(* Logix 5000 project; controller ICA19 vendor 1 type 14 code 150 rev 37.11; software revision 37.00 *)

TASK MainTask (continuous, watchdog 500 ms) : MainProgram

MODULES
   Local : vendor 1 type 14 code 150 (Compact 0, rev 37.11)
      Discrete_IO : Embedded (Compact 1, rev 3.1, Output RPI 20 ms)
      Analog_IO : Embedded (Compact 2, rev 1.1, Output RPI 80 ms)
      Counters : Embedded (Compact 3, rev 1.1, Output RPI 20 ms)
END_MODULES

VAR_GLOBAL   (* controller tags *)
   BottomLimit : ALIAS FOR Local:1:I.Data.1;
   Control : ALIAS FOR Local:1:I.Data.12;
   Door : STRING := 'Door is:';
   DoorClosed : STRING := 'Closed';
   DoorClosing : STRING := ' closing';
   DoorOpened : STRING := ' opening';
   DoorOpening : STRING := 'Opened';
   DoorOut : STRING;
   DoorStopped : STRING := 'stopped';
   MotorDOWN : ALIAS FOR Local:1:O.Data.0;
   MotorStop : ALIAS FOR Local:1:O.Data.2;
   MotorUP : ALIAS FOR Local:1:O.Data.1;
   Safety : STRING;
   SafetyLaser : ALIAS FOR Local:1:I.Data.11;
   SEQ : DINT;
   TopBottom : ALIAS FOR Local:1:I.Data.3;
   TopLimit : ALIAS FOR Local:1:I.Data.2;
END_VAR

PROGRAM MainProgram   (* main routine MainRoutine *)

ROUTINE MainRoutine   (* ladder *)
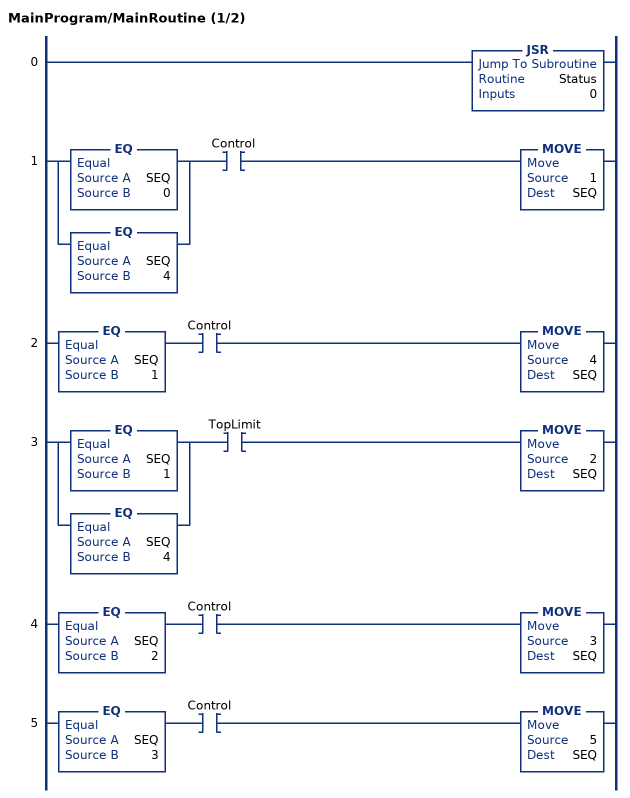
   0: JSR(Status,0);
   1: [EQ(SEQ,0) ,EQ(SEQ,4) ]XIC(Control)MOVE(1,SEQ);
   2: EQ(SEQ,1)XIC(Control)MOVE(4,SEQ);
   3: [EQ(SEQ,1) ,EQ(SEQ,4) ]XIC(TopLimit)MOVE(2,SEQ);
   4: EQ(SEQ,2)XIC(Control)MOVE(3,SEQ);
   5: EQ(SEQ,3)XIC(Control)MOVE(5,SEQ);
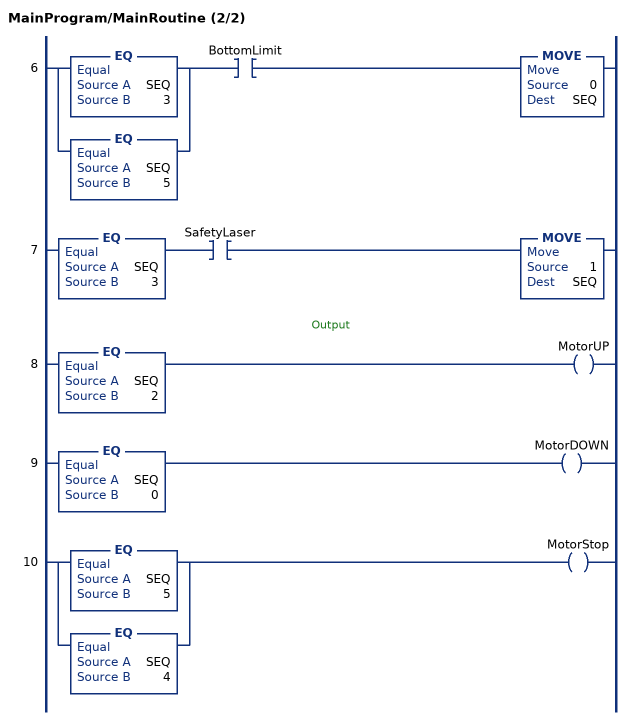
   6: [EQ(SEQ,3) ,EQ(SEQ,5) ]XIC(BottomLimit)MOVE(0,SEQ);
   7: EQ(SEQ,3)XIC(SafetyLaser)MOVE(1,SEQ);
   // Output
   8: EQ(SEQ,2)OTE(MotorUP);
   9: EQ(SEQ,0)OTE(MotorDOWN);
   10: [EQ(SEQ,5) ,EQ(SEQ,4) ]OTE(MotorStop);
END_ROUTINE

ROUTINE Status   (* structured text *)
   if SEQ=0 then
   	concat(Door,DoorClosed,DoorOut);
   end_if;
   
   if SEQ=1 then
   	concat(Door,DoorOpened,DoorOut);
   	end_if;
   
   if SEQ=2 then
   	concat(Door,DoorOpening,DoorOut);
   end_if;
   
   if SEQ=3 then
   	concat(Door,DoorClosing,DoorOut);
   end_if;
   
   if SEQ=5 then
   	concat(Door,DoorStopped,DoorOut);
   end_if;
   
END_ROUTINE
END_PROGRAM
